{attribute 'qualified_only'}
VAR_GLOBAL
	Dynamics AT%Q*: ST_Dynamics;
	Reset : BOOL;
	Run: BOOL;
	SafetyInRun : BOOL; 
	
END_VAR

(* stored: Version 1.1.0.1, ProductVersion 3.1.4026.8
   GVL GVL_DataExchange: Id {9dcb8ac7-c615-4446-ac67-0e2d65200b3f} *)
